FUNCTION F_ChkSettingLimitF : BOOL
VAR_IN_OUT
	fValue		: LREAL;
	stSetting 	: ST_Data_Item;
END_VAR
VAR_OUTPUT
	stInfo 		: ST_Text;
END_VAR

F_ChkSettingLimitF := FALSE;

IF (stSetting.eDataType = E_DataType.eDataType_lreal) AND fValue > stSetting.fValueMax THEN
	stInfo.wsName := "input to high";
	stInfo.wsNameId := "inputtohigh";
	RETURN;
END_IF

IF (stSetting.eDataType = E_DataType.eDataType_lreal) AND fValue < stSetting.fValueMin THEN
	stInfo.wsName := "input to low";
	stInfo.wsNameId := "inputtolow";
	RETURN;
END_IF

IF (stSetting.eDataType = E_DataType.eDataType_time_s) AND fValue > stSetting.fValueMax THEN
	stInfo.wsName := "input to high";
	stInfo.wsNameId := "inputtohigh";
	RETURN;
END_IF

IF (stSetting.eDataType = E_DataType.eDataType_time_s) AND fValue < stSetting.fValueMin THEN
	stInfo.wsName := "input to low";
	stInfo.wsNameId := "inputtolow";
	RETURN;
END_IF

IF (stSetting.eDataType = E_DataType.eDataType_time_m) AND fValue > stSetting.fValueMax THEN
	stInfo.wsName := "input to high";
	stInfo.wsNameId := "inputtohigh";
	RETURN;
END_IF

IF (stSetting.eDataType = E_DataType.eDataType_time_m) AND fValue < stSetting.fValueMin THEN
	stInfo.wsName := "input to low";
	stInfo.wsNameId := "inputtolow";
	RETURN;
END_IF

IF (stSetting.eDataType = E_DataType.eDataType_time_h) AND fValue > stSetting.fValueMax THEN
	stInfo.wsName := "input to high";
	stInfo.wsNameId := "inputtohigh";
	RETURN;
END_IF

IF (stSetting.eDataType = E_DataType.eDataType_time_h) AND fValue < stSetting.fValueMin THEN
	stInfo.wsName := "input to low";
	stInfo.wsNameId := "inputtolow";
	RETURN;
END_IF

F_ChkSettingLimitF := TRUE;

END_FUNCTION

(* stored: Version 1.1.0.1, ProductVersion 3.1.4024.12
   POU F_ChkSettingLimitF: Id {94eb53f6-26f7-499b-9895-fe8bdaa871b8}, SpecialFunc None *)
